PROGRAM MAIN
VAR
	_sampleComponentTests : SampleComponentTests;
END_VAR

END_PROGRAM

(* stored: Version 1.1.0.1, ProductVersion 3.1.4024.9
   POU MAIN: Id {d440c2ad-ecd0-096f-265b-7a11e8982c80}, SpecialFunc None *)
